FUNCTION_BLOCK FB_WashingMachine

VAR_IN_OUT
	stWash : ST_Wash;
END_VAR
VAR
	iWashStrategy : I_WashStrategy;
	iMotor : I_Motor;
	iWaterController : I_WaterController;
	
	eMachineState : E_MachineState;
	tTotalTime : TIME ;
	bRunning : BOOL;
	tBaseTime : TIME := T#5S;
	nRinseCount : INT;
	
	fbTimer : TON ;
	
END_VAR


IF tTotalTime <> T#0S THEN
	fbTimer (IN := bRunning , PT := tTotalTime);
END_IF

IF __ISVALIDREF(stWash) THEN
	
	CASE eMachineState OF
		E_MachineState.IDLE:
			bRunning := Start();
			eMachineState := E_MachineState.CONFIGURING;
			
			
		E_MachineState.CONFIGURING:
			nRinseCount := 0;
			iWashStrategy := SelectStrategy();
			iMotor := SelectMotor();
			iWaterController := SelectWaterController();
			IF iWashStrategy <> 0 AND iWaterController <> 0 AND iMotor <> 0 THEN
				tTotalTime := iWaterController.GetDuration(stWash) * iWashStrategy.GetRinseCount() + iWashStrategy.GetDuration();
				eMachineState := E_MachineState.FILLING;
			ELSE
				eMachineState := E_MachineState.ERROR;
			END_IF
		
		E_MachineState.FILLING:
			IF iWaterController.StartFill() THEN
				eMachineState := E_MachineState.WASHING;
			END_IF
				
		E_MachineState.WASHING:
			IF iWashStrategy.StartWash(iMotor) THEN
				eMachineState := E_MachineState.DRAINING;
			END_IF
		
		E_MachineState.DRAINING:
				IF NOT iWaterController.StartDrain() THEN
					nRinseCount := nRinseCount + 1;
					IF nRinseCount = iWashStrategy.GetRinseCount() THEN
						eMachineState := E_MachineState.DRYING;
					ELSE
						eMachineState := E_MachineState.FILLING;
					END_IF
				END_IF
		E_MachineState.DRYING:
			IF iWashStrategy.StartSpin() THEN
				eMachineState := E_MachineState.COMPLETED;
			END_IF
			
			E_MachineState.COMPLETED:
			bRunning := FALSE;
			fbTimer( IN := bRunning);
			
		E_MachineState.ERROR:
		
		
	END_CASE
	
END_IF

PROPERTY eState : E_MachineState
GET
eState := eMachineState;
END_GET
SET // PRIVATE
eMachineState := eState;
END_SET
END_PROPERTY

METHOD SelectMotor : I_Motor
VAR_INPUT
END_VAR
SelectMotor := GVL_References.fbMotor;
END_METHOD

METHOD PRIVATE SelectStrategy : I_WashStrategy
VAR_INPUT
END_VAR
VAR
	
END_VAR
CASE stWash.eWashStrategy OF
	E_Strategy.SOFT :
	SelectStrategy :=  GVL_References.fbSoftWash;
	
	E_Strategy.NORMAL :
	SelectStrategy :=  GVL_References.fbNormalWash;
	
	E_Strategy.HARD :
	SelectStrategy :=  GVL_References.fbHeavyWash;
	
END_CASE
END_METHOD

METHOD SelectWaterController : I_WaterController
VAR_INPUT
END_VAR
SelectWaterController :=  GVL_References.fbWaterController;
END_METHOD

METHOD Start : BOOL
VAR_INPUT
END_VAR
Start := TRUE;
END_METHOD

METHOD Stop : BOOL
VAR_INPUT
END_VAR
END_METHOD

PROPERTY tRemainingTime : TIME
GET
tRemainingTime := tTotalTime - fbTimer.ET;
END_GET
SET // PRIVATE
tTotalTime := tRemainingTime;
END_SET
END_PROPERTY

END_FUNCTION_BLOCK

(* stored: Version 1.1.0.1, ProductVersion 3.1.4024.16
   POU FB_WashingMachine: Id {533b8205-1e07-4998-827d-1f3b127b70ad}, SpecialFunc None
   Property eState: Id {9eb26405-ab77-4215-9e4b-5261859df458}
   Get Get: Id {75450bf7-8a2e-4da7-bf7a-4c0318bbb720}
   Set Set: Id {0a692673-5a45-4181-a89f-b89da7cd827c}
   Method SelectMotor: Id {ca951e7e-739c-49fb-acab-b80aa14296a5}
   Method SelectStrategy: Id {6ef3cceb-1fa2-4f2e-af62-8c5ba15a6afb}
   Method SelectWaterController: Id {96fd3fe0-7873-43ae-a291-313852a54e2c}
   Method Start: Id {d04ebe96-dff9-4b6d-8e28-83c84e090aa8}
   Method Stop: Id {eedaa334-e689-4c2e-9e59-a00d7921cfb5}
   Property tRemainingTime: Id {2ae82297-0e7a-47c1-bf6f-19f0329c494b}
   Get Get: Id {008e38d0-36e6-4810-b6c3-8a0942dcf1d6}
   Set Set: Id {d8e58f91-fb47-41b8-be75-38907c1b1b1d} *)
